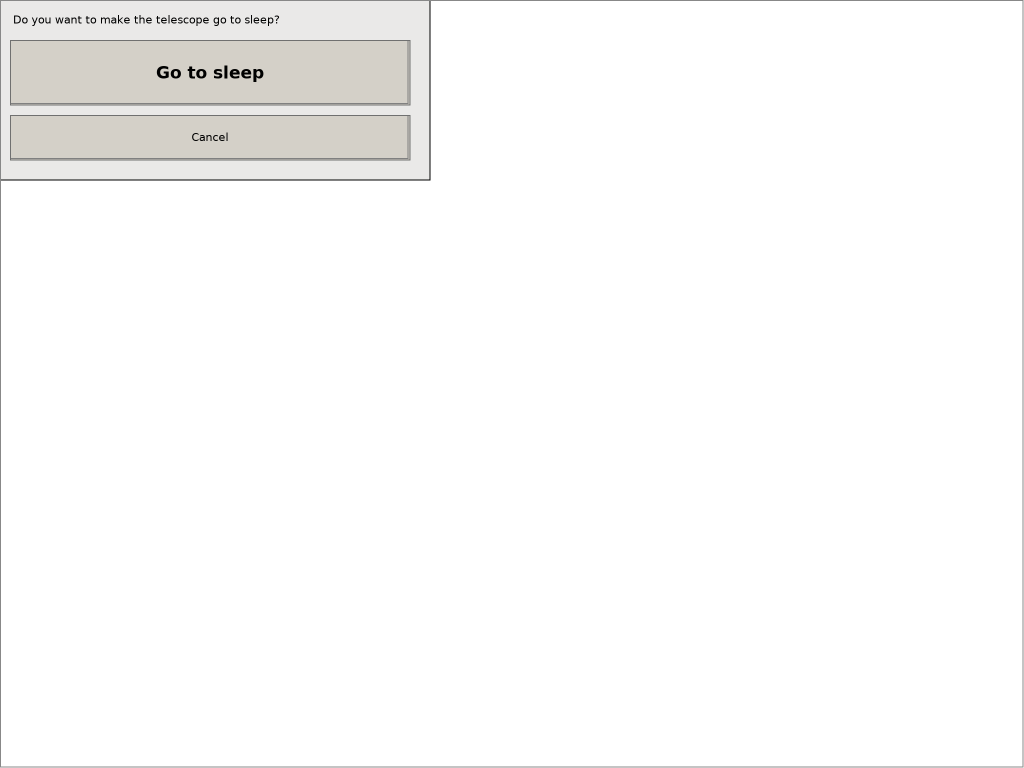
VISUALIZATION VISU_MTCSGoToSleepDialog  // 1024x768
    Rectangle (0,0 430x180)
    Button (10,40 400x65), "Go to sleep", input disabled if: GLOBAL.mtcs.processes.goToSleep.statuses.enabledStatus.disabled
        OnMouseClick: execute { GLOBAL.mtcs.processes.goToSleep.do_request := TRUE; }
        OnMouseClick: CloseDialog Dialog=VISU_MTCSGoToSleepDialog, Result=OK, NumpadKeypadSet=True
    Button (10,115 400x45), "Cancel"
        OnMouseClick: CloseDialog Dialog=VISU_MTCSGoToSleepDialog, Result=OK, NumpadKeypadSet=True
    Label (10,5 400x30), "Do you want to make the telescope go to sleep?"
END_VISUALIZATION

(* stored: Version 1.1.0.1, ProductVersion 3.1.4018.5
   Visu VISU_MTCSGoToSleepDialog: Id {d501b4d2-de97-4c1d-9032-cb001c6cf7a7} *)
